FUNCTION_BLOCK Service_DIMeasure (* Basic Function Block Type *)
  (* Standard: 61499-2 *)
  (* Version 0.0, 2014-5-4, wildai, nxtControl GmbH, Template *)
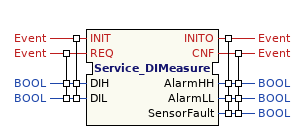
  EVENT_INPUT
    INIT WITH DIH, DIL; (* Initialization Request *)
    REQ WITH DIH, DIL; (* Normal Execution Request *)
  END_EVENT
  EVENT_OUTPUT
    INITO WITH AlarmHH, AlarmLL, SensorFault; (* Initialization Confirm *)
    CNF WITH AlarmHH, AlarmLL, SensorFault; (* Execution Confirmation *)
  END_EVENT
  VAR_INPUT
    DIH : BOOL;
    DIL : BOOL;
  END_VAR
  VAR_OUTPUT
    AlarmHH : BOOL;
    AlarmLL : BOOL;
    SensorFault : BOOL;
  END_VAR
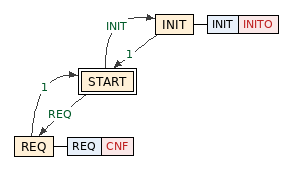
  EC_STATES
    START; (* Initial State *)
    INIT : INIT -> INITO; (* Initialization *)
    REQ : REQ -> CNF; (* Normal execution *)
  END_STATES
  EC_TRANSITIONS
    START TO INIT := INIT;
    INIT TO START := 1;
    START TO REQ := REQ;
    REQ TO START := 1;
  END_TRANSITIONS
  ALGORITHM INIT IN ST: (* Initialization algorithm *)
;

SensorFault := FALSE;
AlarmHH := FALSE;
AlarmLL := FALSE;
  END_ALGORITHM
  ALGORITHM REQ IN ST: (* Normally executed algorithm *)
;
IF DIH AND DIL THEN
	SensorFault := TRUE;
	AlarmHH := FALSE;
	AlarmLL := FALSE;
ELSE
	SensorFault := FALSE;
	IF DIH THEN
		AlarmHH := TRUE;
		AlarmLL := FALSE;
	ELSIF DIL THEN
		AlarmHH := FALSE;
		AlarmLL := TRUE;
	ELSE
		AlarmHH := FALSE;
		AlarmLL := FALSE;
	END_IF;
END_IF;
  END_ALGORITHM
END_FUNCTION_BLOCK
